# EPICS StreamDevice protocol: Switch.proto
##################################################
# General Settings
##################################################

Terminator = CR;
ReplyTimeout = 1000;
locktimeout = 5000;
readtimeout  = 1000;
extrainput   = Ignore;

###################################################
# Get functions
###################################################

# Read IDN from Switch
getIDN {
   out "*IDN?";
   in "%s";
}

# Read State
getState {
   out ":clos:stat?";
   in "(@%39c";
}

getStatewf {
   separator=",";
   in "array = (%s)";
}

# Set Memory Recall
setMemRecall{
   out ":MEM:RECALL M%i";
}

# Set Display Front
setFrontDisplay{
   out ":DISP:WIND2:TEXT:STAT ON";
}

# Set Memory Location
setMemoryLoc {
   out ":DISP:WIND2:TEXT:DATA 'mem location  %i\'";
}
